{attribute 'GeneratedUsingTerminal: EL9576-0000-0020'}
{attribute addProperty BoxType "EL9576-0000-0020"}
{attribute addProperty Id "BCT_InputsAT %I*BCT_Inputs_8B1D510C16WcStateAT %I*WcState_9091E0EB2InfoDataAT %I*InfoData_94A18F5E2"}
{attribute addProperty CRC "2936953898"}
{attribute addProperty Size "20"}
TYPE EL9576_AF0E5C2A EXTENDS EtcSlaveTerminalBase_947E5A46 :
STRUCT
	{attribute addProperty Name "BCT_Inputs"}
	BCT_Inputs : BCT_Inputs_8B1D510C;
	{attribute addProperty Name "WcState"}
	WcState : WcState_9091E0EB;
	{attribute addProperty Name "InfoData"}
	InfoData : InfoData_94A18F5E;
END_STRUCT
END_TYPE

(* stored: Version 1.2.0.0, ProductVersion 3.1.4024.9
   DUT EL9576_AF0E5C2A: Id {1fc09f91-6fb1-4f5b-ba36-4695467afadf} *)
